# EPICS substitutions: rsaApp/Db/userHost.substitutions
# Example substitutions file

file "db/dbExample1.db" {
    { user = "joaoHost" }
}

file db/dbExample2.db {
    pattern { user, no, scan }
        { "joaoHost", 1, "1 second" }
        { "joaoHost", 2, "2 second" }
        { "joaoHost", 3, "5 second" }
}
